PROGRAM PRG_TEST
VAR
	suite_Example : Example;
END_VAR

TcUnit.RUN();

END_PROGRAM

(* stored: Version 1.1.0.1, ProductVersion 3.1.4024.12
   POU PRG_TEST: Id {05bea583-3305-4137-8317-3c4e75dfa876}, SpecialFunc None *)
